// TIA Portal V19 export
FUNCTION_BLOCK "FB_ManageDoor"   // FB1010, LAD
{ S7_Optimized_Access := 'TRUE' }
// stored: AutoNumber false, MemoryReserve 100, SetENOAutomatically false
   VAR_INPUT
      nMode { ExternalAccessible := 'False'; ExternalVisible := 'False'; ExternalWritable := 'False'} : Int;
      xSafetyState { ExternalAccessible := 'False'; ExternalVisible := 'False'; ExternalWritable := 'False'} : Bool;
      xDoorClosed { ExternalAccessible := 'False'; ExternalVisible := 'False'; ExternalWritable := 'False'} : Bool;   // ON when the door is closed
      xBoldTongueInserted { ExternalAccessible := 'False'; ExternalVisible := 'False'; ExternalWritable := 'False'} : Bool;   // Bolt tongue inserted into the evaluation module
      xGuardLocked { ExternalAccessible := 'False'; ExternalVisible := 'False'; ExternalWritable := 'False'} : Bool;   // Guard locking solenoid in locked position
      xPBAccesReq { ExternalAccessible := 'False'; ExternalVisible := 'False'; ExternalWritable := 'False'} : Bool;
      xPBLockDoor { ExternalAccessible := 'False'; ExternalVisible := 'False'; ExternalWritable := 'False'} : Bool;
      xRobotStopped { ExternalAccessible := 'False'; ExternalVisible := 'False'; ExternalWritable := 'False'} : Bool;
      xCellStopped { ExternalAccessible := 'False'; ExternalVisible := 'False'; ExternalWritable := 'False'} : Bool;
      xTestLamp { ExternalAccessible := 'False'; ExternalVisible := 'False'; ExternalWritable := 'False'} : Bool;
      xPulseBit { ExternalAccessible := 'False'; ExternalVisible := 'False'; ExternalWritable := 'False'} : Bool;
   END_VAR
   VAR_OUTPUT
      xLockDoor { ExternalAccessible := 'False'; ExternalVisible := 'False'; ExternalWritable := 'False'} : Bool;
      xUnlockDoor { ExternalAccessible := 'False'; ExternalVisible := 'False'; ExternalWritable := 'False'} : Bool;
      xResetDoor { ExternalAccessible := 'False'; ExternalVisible := 'False'; ExternalWritable := 'False'} : Bool;
      xStopReq { ExternalAccessible := 'False'; ExternalVisible := 'False'; ExternalWritable := 'False'} : Bool;
      xLightAccesReq { ExternalAccessible := 'False'; ExternalVisible := 'False'; ExternalWritable := 'False'} : Bool;
      xLightLockDoor { ExternalAccessible := 'False'; ExternalVisible := 'False'; ExternalWritable := 'False'} : Bool;
   END_VAR
   VAR
      sFPAccesReq { ExternalAccessible := 'False'; ExternalVisible := 'False'; ExternalWritable := 'False'} : Bool;
      sxAccesRequested { ExternalAccessible := 'False'; ExternalVisible := 'False'; ExternalWritable := 'False'} : Bool;
      sxAccesAllowed { ExternalAccessible := 'False'; ExternalVisible := 'False'; ExternalWritable := 'False'} : Bool;
   END_VAR
   VAR_TEMP
      tAccesReq : Bool;
   END_VAR
   VAR CONSTANT
      ModeAuto : Int := 1;
      ModeManu : Int := 2;
      ModeMaintenance : Int := 3;
   END_VAR
   VAR_TEMP   // added for the SCL form of the ladder/FBD networks
      _w1 : Bool;
      _w2 : Bool;
   END_VAR
BEGIN

REGION Network 1: Set and Reset internal acces request
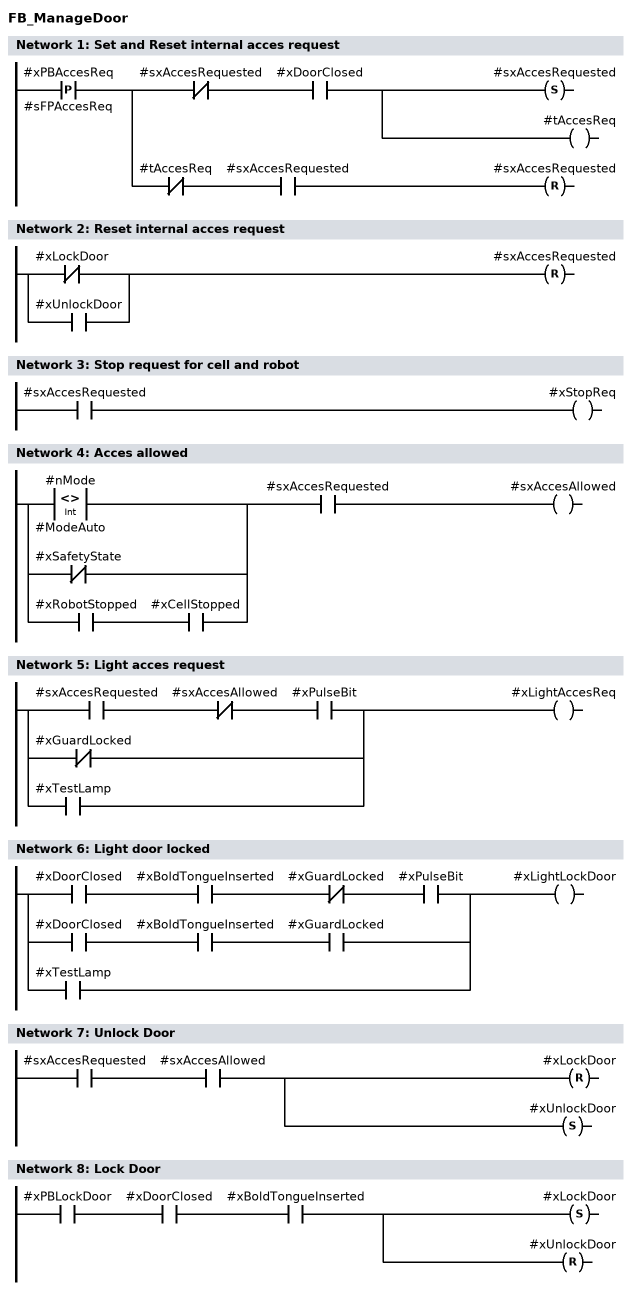
   RUNG wire#powerrail
      P_Contact(operand := #xPBAccesReq, bit := #sFPAccesReq)
      wire#w1
      I_Contact( #sxAccesRequested )
      Contact( #xDoorClosed )
      wire#w2
      S_Coil( #sxAccesRequested )
   END_RUNG
   RUNG wire#w2
      Coil( #tAccesReq )
   END_RUNG
   RUNG wire#w1
      I_Contact( #tAccesReq )
      Contact( #sxAccesRequested )
      R_Coil( #sxAccesRequested )
   END_RUNG
   // the same network as SCL:
   #_w1 := #xPBAccesReq AND NOT #sFPAccesReq;   // rising edge of #xPBAccesReq
   #sFPAccesReq := #xPBAccesReq;
   #_w2 := #_w1 AND NOT #sxAccesRequested AND #xDoorClosed;
   IF #_w2 THEN #sxAccesRequested := TRUE; END_IF;
   #tAccesReq := #_w2;
   IF #_w1 AND NOT #tAccesReq AND #sxAccesRequested THEN #sxAccesRequested := FALSE; END_IF;
END_REGION

REGION Network 2: Reset internal acces request
   RUNG wire#powerrail
      I_Contact( #xLockDoor )
      wire#w1
      R_Coil( #sxAccesRequested )
   END_RUNG
   RUNG wire#powerrail
      Contact( #xUnlockDoor )
   END_RUNG wire#w1
   // the same network as SCL:
   IF NOT #xLockDoor OR #xUnlockDoor THEN #sxAccesRequested := FALSE; END_IF;
END_REGION

REGION Network 3: Stop request for cell and robot
   RUNG wire#powerrail
      Contact( #sxAccesRequested )
      Coil( #xStopReq )
   END_RUNG
   // the same network as SCL:
   #xStopReq := #sxAccesRequested;
END_REGION

REGION Network 4: Acces allowed
   RUNG wire#powerrail
      { S7_Templates := "SrcType := Int" } NE_Contact(in1 := #nMode, in2 := #ModeAuto)
      wire#w1
      Contact( #sxAccesRequested )
      Coil( #sxAccesAllowed )
   END_RUNG
   RUNG wire#powerrail
      I_Contact( #xSafetyState )
   END_RUNG wire#w1
   RUNG wire#powerrail
      Contact( #xRobotStopped )
      Contact( #xCellStopped )
   END_RUNG wire#w1
   // the same network as SCL:
   #sxAccesAllowed := ((#nMode <> #ModeAuto) OR NOT #xSafetyState OR (#xRobotStopped AND #xCellStopped)) AND #sxAccesRequested;
END_REGION

REGION Network 5: Light acces request
   RUNG wire#powerrail
      Contact( #sxAccesRequested )
      I_Contact( #sxAccesAllowed )
      Contact( #xPulseBit )
      wire#w1
      Coil( #xLightAccesReq )
   END_RUNG
   RUNG wire#powerrail
      I_Contact( #xGuardLocked )
   END_RUNG wire#w1
   RUNG wire#powerrail
      Contact( #xTestLamp )
   END_RUNG wire#w1
   // the same network as SCL:
   #xLightAccesReq := (#sxAccesRequested AND NOT #sxAccesAllowed AND #xPulseBit) OR NOT #xGuardLocked OR #xTestLamp;
END_REGION

REGION Network 6: Light door locked
   RUNG wire#powerrail
      Contact( #xDoorClosed )
      Contact( #xBoldTongueInserted )
      I_Contact( #xGuardLocked )
      Contact( #xPulseBit )
      wire#w1
      Coil( #xLightLockDoor )
   END_RUNG
   RUNG wire#powerrail
      Contact( #xDoorClosed )
      Contact( #xBoldTongueInserted )
      Contact( #xGuardLocked )
   END_RUNG wire#w1
   RUNG wire#powerrail
      Contact( #xTestLamp )
   END_RUNG wire#w1
   // the same network as SCL:
   #xLightLockDoor := (#xDoorClosed AND #xBoldTongueInserted AND NOT #xGuardLocked AND #xPulseBit) OR (#xDoorClosed AND #xBoldTongueInserted AND #xGuardLocked) OR #xTestLamp;
END_REGION

REGION Network 7: Unlock Door
   RUNG wire#powerrail
      Contact( #sxAccesRequested )
      Contact( #sxAccesAllowed )
      wire#w1
      R_Coil( #xLockDoor )
   END_RUNG
   RUNG wire#w1
      S_Coil( #xUnlockDoor )
   END_RUNG
   // the same network as SCL:
   IF #sxAccesRequested AND #sxAccesAllowed THEN
       #xLockDoor := FALSE;
       #xUnlockDoor := TRUE;
   END_IF;
END_REGION

REGION Network 8: Lock Door
   RUNG wire#powerrail
      Contact( #xPBLockDoor )
      Contact( #xDoorClosed )
      Contact( #xBoldTongueInserted )
      wire#w1
      S_Coil( #xLockDoor )
   END_RUNG
   RUNG wire#w1
      R_Coil( #xUnlockDoor )
   END_RUNG
   // the same network as SCL:
   IF #xPBLockDoor AND #xDoorClosed AND #xBoldTongueInserted THEN
       #xLockDoor := TRUE;
       #xUnlockDoor := FALSE;
   END_IF;
END_REGION
END_FUNCTION_BLOCK
